TYPE ST_AddStationDoubleData :
STRUCT
	sObjectID					: STRING := 'MAIN.fbMMServer';
	sMethodID					: STRING := 'MAIN.fbMMServer#M_AddStationDouble';
	iStatus						: INT;
	iNoOfInputArgs				: BYTE := 10;
	iNoOfOutputArgs				: BYTE := 2;
	stInput						: ST_AddStationDoubleDataIn;
	stOutput					: ST_AddStationDoubleDataOut;	
END_STRUCT
END_TYPE

(* stored: Version 1.1.0.1, ProductVersion 3.1.4024.5
   DUT ST_AddStationDoubleData: Id {0fa124af-a801-4715-8b48-81f0ee51f21d} *)
